PROGRAM MAIN
VAR
	counter : INT;
	testDeleteIfDontWork : bool;
END_VAR

counter := counter + 1;

IF counter = 100 THEN
	counter := 0;
END_IF

END_PROGRAM

(* stored: Version 1.1.0.1, ProductVersion 3.1.4024.13
   POU MAIN: Id {76ab99c2-600b-41ce-824f-f20e8be30e39}, SpecialFunc None *)
